FUNCTION_BLOCK FeedReactor1PBasic (* Basic Function Block Type *)
  (* Standard: 61499-2 *)
  (* Version 0.0, 6/15/2026, Schneider Electric, Template *)
  PACKAGE SE.Nereda;
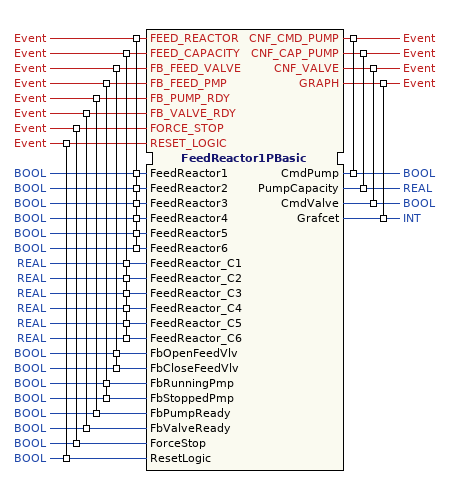
  EVENT_INPUT
    FEED_REACTOR WITH FeedReactor1, FeedReactor2, FeedReactor3, FeedReactor4, FeedReactor5, FeedReactor6;
    FEED_CAPACITY WITH FeedReactor_C1, FeedReactor_C2, FeedReactor_C3, FeedReactor_C4, FeedReactor_C5, FeedReactor_C6;
    FB_FEED_VALVE WITH FbOpenFeedVlv, FbCloseFeedVlv;
    FB_FEED_PMP WITH FbRunningPmp, FbStoppedPmp;
    FB_PUMP_RDY WITH FbPumpReady;
    FB_VALVE_RDY WITH FbValveReady;
    FORCE_STOP WITH ForceStop;
    RESET_LOGIC WITH ResetLogic;
  END_EVENT
  EVENT_OUTPUT
    CNF_CMD_PUMP WITH CmdPump;
    CNF_CAP_PUMP WITH PumpCapacity;
    CNF_VALVE WITH CmdValve;
    GRAPH WITH Grafcet;
  END_EVENT
  VAR_INPUT
    FeedReactor1 : BOOL;
    FeedReactor2 : BOOL;
    FeedReactor3 : BOOL;
    FeedReactor4 : BOOL;
    FeedReactor5 : BOOL;
    FeedReactor6 : BOOL;
    FeedReactor_C1 : REAL;
    FeedReactor_C2 : REAL;
    FeedReactor_C3 : REAL;
    FeedReactor_C4 : REAL;
    FeedReactor_C5 : REAL;
    FeedReactor_C6 : REAL;
    FbOpenFeedVlv : BOOL;
    FbCloseFeedVlv : BOOL;
    FbRunningPmp : BOOL;
    FbStoppedPmp : BOOL;
    FbPumpReady : BOOL;
    FbValveReady : BOOL;
    ForceStop : BOOL;
    ResetLogic : BOOL;
  END_VAR
  VAR_OUTPUT
    CmdPump : BOOL;
    PumpCapacity : REAL;
    CmdValve : BOOL;
    Grafcet : INT;
  END_VAR
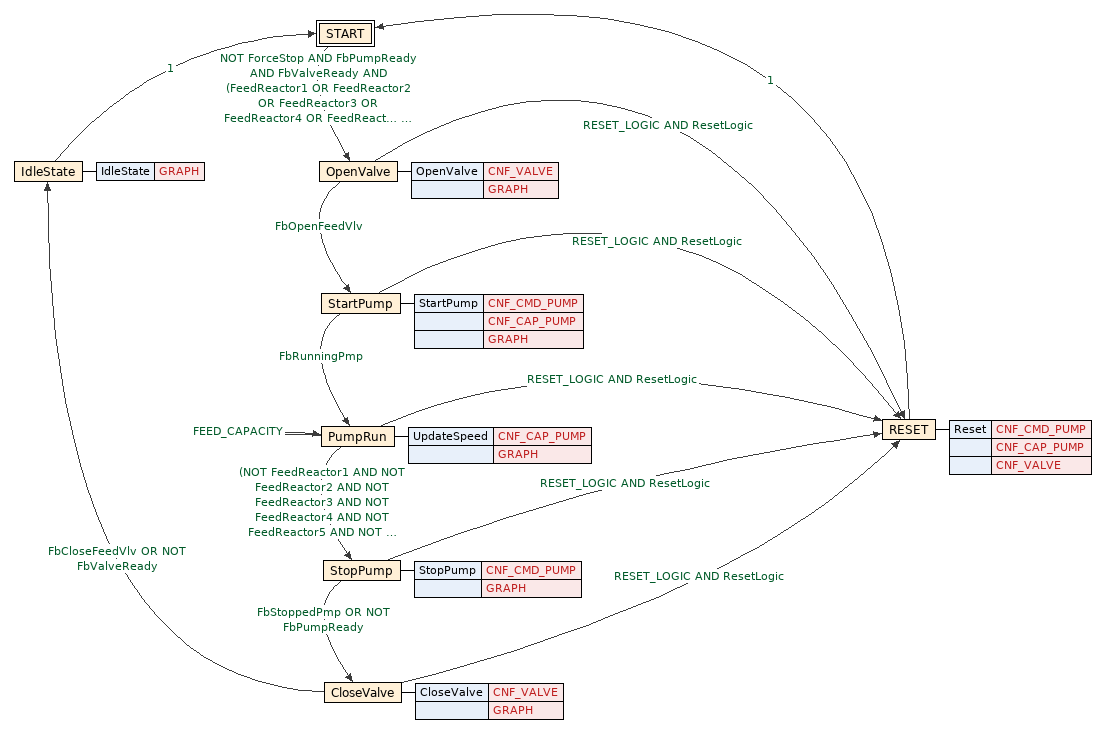
  EC_STATES
    START; (* Initial State *)
    OpenValve : OpenValve -> CNF_VALVE, -> GRAPH;
    StartPump : StartPump -> CNF_CMD_PUMP, -> CNF_CAP_PUMP, -> GRAPH;
    PumpRun : UpdateSpeed -> CNF_CAP_PUMP, -> GRAPH;
    StopPump : StopPump -> CNF_CMD_PUMP, -> GRAPH;
    CloseValve : CloseValve -> CNF_VALVE, -> GRAPH;
    RESET : Reset -> CNF_CMD_PUMP, -> CNF_CAP_PUMP, -> CNF_VALVE;
    IdleState : IdleState -> GRAPH;
  END_STATES
  EC_TRANSITIONS
    START TO OpenValve := NOT ForceStop AND FbPumpReady AND FbValveReady AND (FeedReactor1 OR FeedReactor2 OR FeedReactor3 OR FeedReactor4 OR FeedReactor5 OR FeedReactor6);
    OpenValve TO StartPump := FbOpenFeedVlv;
    StartPump TO PumpRun := FbRunningPmp;
    PumpRun TO StopPump := (NOT FeedReactor1 AND NOT FeedReactor2 AND NOT FeedReactor3 AND NOT FeedReactor4 AND NOT FeedReactor5 AND NOT FeedReactor6) OR ForceStop OR NOT FbPumpReady OR NOT FbValveReady;
    StopPump TO CloseValve := FbStoppedPmp OR NOT FbPumpReady;
    CloseValve TO IdleState := FbCloseFeedVlv OR NOT FbValveReady;
    PumpRun TO PumpRun := FEED_CAPACITY;
    OpenValve TO RESET := RESET_LOGIC AND ResetLogic;
    StartPump TO RESET := RESET_LOGIC AND ResetLogic;
    PumpRun TO RESET := RESET_LOGIC AND ResetLogic;
    StopPump TO RESET := RESET_LOGIC AND ResetLogic;
    CloseValve TO RESET := RESET_LOGIC AND ResetLogic;
    RESET TO START := 1;
    IdleState TO START := 1;
  END_TRANSITIONS
  ALGORITHM OpenValve IN ST:
;
Grafcet := 1;
CmdValve := TRUE;
  END_ALGORITHM
  ALGORITHM StartPump IN ST:
;
Grafcet := 2;
CmdPump := TRUE;

// Default value
PumpCapacity := 0.0;

// Reactor 1 active
IF FeedReactor1 THEN
	PumpCapacity := FeedReactor_C1;
END_IF;

// Reactor 2 active: keep the highest capacity
IF FeedReactor2 AND (FeedReactor_C2 > PumpCapacity) THEN
	PumpCapacity := FeedReactor_C2;
END_IF;

// Reactor 3 active: keep the highest capacity
IF FeedReactor3 AND (FeedReactor_C3 > PumpCapacity) THEN
	PumpCapacity := FeedReactor_C3;
END_IF;

// Reactor 4 active: keep the highest capacity
IF FeedReactor4 AND (FeedReactor_C4 > PumpCapacity) THEN
	PumpCapacity := FeedReactor_C4;
END_IF;

// Reactor 5 active: keep the highest capacity
IF FeedReactor5 AND (FeedReactor_C5 > PumpCapacity) THEN
	PumpCapacity := FeedReactor_C5;
END_IF;

// Reactor 6 active: keep the highest capacity
IF FeedReactor6 AND (FeedReactor_C6 > PumpCapacity) THEN
	PumpCapacity := FeedReactor_C6;
END_IF;
  END_ALGORITHM
  ALGORITHM UpdateSpeed IN ST:
;
Grafcet := 3;

// Default value
PumpCapacity := 0.0;

// Reactor 1 active
IF FeedReactor1 THEN
	PumpCapacity := FeedReactor_C1;
END_IF;

// Reactor 2 active: keep the highest capacity
IF FeedReactor2 AND (FeedReactor_C2 > PumpCapacity) THEN
	PumpCapacity := FeedReactor_C2;
END_IF;

// Reactor 3 active: keep the highest capacity
IF FeedReactor3 AND (FeedReactor_C3 > PumpCapacity) THEN
	PumpCapacity := FeedReactor_C3;
END_IF;

// Reactor 4 active: keep the highest capacity
IF FeedReactor4 AND (FeedReactor_C4 > PumpCapacity) THEN
	PumpCapacity := FeedReactor_C4;
END_IF;

// Reactor 5 active: keep the highest capacity
IF FeedReactor5 AND (FeedReactor_C5 > PumpCapacity) THEN
	PumpCapacity := FeedReactor_C5;
END_IF;

// Reactor 6 active: keep the highest capacity
IF FeedReactor6 AND (FeedReactor_C6 > PumpCapacity) THEN
	PumpCapacity := FeedReactor_C6;
END_IF;
  END_ALGORITHM
  ALGORITHM StopPump IN ST:
;
Grafcet := 4;
CmdPump := FALSE;
  END_ALGORITHM
  ALGORITHM CloseValve IN ST:
;
Grafcet := 5;
CmdValve := FALSE;
  END_ALGORITHM
  ALGORITHM Reset IN ST:
;
CmdValve := FALSE;
CmdPump := FALSE;
PumpCapacity := 0;
  END_ALGORITHM
  ALGORITHM IdleState IN ST:
;
Grafcet := 6;
  END_ALGORITHM
END_FUNCTION_BLOCK
